REGION Network 1: Block description — Sections 1 to 2
   // ▄▄▄▄▄▄▄▄▄▄▄▄▄▄▄▄▄▄▄▄▄▄▄▄▄▄▄▄▄▄▄▄▄  ＳＴＡＮＤＡＲＤ  ▄▄ 
   // 
   // 
   // TITLE:    DEVICE DRIVER — THREE-WAY VALVE
   // 
   // 
   // ▀▀▀▀▀▀▀▀▀▀▀▀▀▀▀▀▀▀▀▀▀▀▀▀▀▀▀▀▀▀▀▀▀▀▀▀▀▀▀▀▀▀▀▀ 
   // 
   // ┌──────────────────────────────────────────┐
   // │                                          │
   // │          FC11011 — SOFTWARE MODULE DESIGN SPECIFICATION (SMDS)            │
   // │                                          │
   // │      The PDF version of the SMDS for this module is available online here:        │
   // │              https://psop.uk/pal-smds-fc11011-p               │
   // │                                          │
   // │      It is also available as part of the Project User Defined Documentation,      │
   // │      it can be accessed by selecting this module in the Project Tree          │
   // │      (on the left) and pressing SHIFT+F1                        │
   // │                                          │
   // └─────────────────────────────────────── ʷᴵᴰ⁻ᵇᶠᵍ  ┘
   // 
   // FC11011_StdDevValve3Way controls the operation of 3-way valve with a common energised port 
   // (the action of the valve switches the common port to one of the other two ports) configured with 
   // either position feedback or no position feedback.
   // 
   // The module supports automatic and manual control and can be configured with simulation mode 
   // to allow the valve limit switch signals to be overwritten and set to follow the demand output. 
   // 
   // The module generates fault logic for the valve that will trigger specific alarms depending on the 
   // fault in question. The alarms within this block are: 
   // 
   //    •   Failed to Energise 
   // 
   //    •   Failed to Deenergise 
   // 
   //    •   Failed while Energised
   // 
   //    •   Failed while Deenergised
   // 
   //    •   External Fault 
   // 
   // Separate operation times for energising and deenergising can be defined. 
   // 
   // The valve module supports all forms of interlock, permissive and trip signals, and emergency stop 
   // signals. The module has the conditional facility to allow the operator to bypass interlocks, 
   // permissive and trip conditions.
   // 
   // Various status signals are generated for supervisory systems:
   // 
   //    •   Deenergised
   // 
   //    •   Energising
   // 
   //    •   Energised
   // 
   //    •   Deenergising
   // 
   //    •   Fault
   // 
   // The module also generates status signals for the selected operating modes and conditions.
   // 
   // 
   // ▄▄▄▄▄▄▄▄▄▄▄▄▄▄▄▄▄▄▄▄▄▄▄▄▄▄▄▄▄▄▄▄▄▄▄▄▄▄▄▄▄▄▄▄
   // 1.     BLOCK TECHNICAL SUMMARY
   // 
   // 
   //  ――――――――――――――――――――――――――――――――――――――――――
   //  NOMENCLATURE & ADDRESSING
   //  ――――――――――――――――――――――――――――――――――――――――――
   //  BLOCK TITLE         Three-way Valve
   //  BLOCK FUNCTION GROUP    Device Driver 
   //  BLOCK ADDRESS       FC11011
   //  BLOCK SYMBOL        FC11011_StdDevValve3Way
   //  BLOCK USER ID         StdDevValve3Way
   // 
   //  ――――――――――――――――――――――――――――――――――――――――――
   //  BLOCK TYPE & USAGE
   //  ――――――――――――――――――――――――――――――――――――――――――
   //  BLOCK TYPE         Function (FC)
   //  BLOCK NUMBER        11011
   //  LANGUAGE           LAD
   //  OPTIMISED ACCESS     Yes
   //  PAL USAGE TYPE       Standard block
   // 
   //  ――――――――――――――――――――――――――――――――――――――――――
   //  METRICS
   //  ――――――――――――――――――――――――――――――――――――――――――
   //  EXECUTION TIME       66.5 μs¹
   //  LOAD MEMORY       98.6 kB
   //  WORK MEMORY           2.1 kB  
   //  ――――――――――――――――――――――――――――――――――――――――――
   //                ¹ Measured on: CPU-1515-2PN (order no. 6ES7512-2AM02-0AB0) 
   //                             https://psop.uk/pal-ds-cpu1515
   // 
   // 
   // 
   // ▂▂▂▂▂▂▂▂▂▂▂▂▂▂▂▂▂▂▂▂▂▂▂▂▂▂▂▂▂▂▂▂▂▂▂▂▂▂▂▂▂▂▂▂
   // 1.1      Additional document references
   // 
   // 
   // Only those documents specified in OB1 (section DOCUMENT REFERENCES) are listed within this 
   // block. There are no additional document references.
   // 
   //                ━━━   ⬙⬙⬙⬙⬙⬙   ━━━
   // 
   // 
   // 
   // ▄▄▄▄▄▄▄▄▄▄▄▄▄▄▄▄▄▄▄▄▄▄▄▄▄▄▄▄▄▄▄▄▄▄▄▄▄▄▄▄▄▄▄▄
   // 2.     FUNCTIONAL DESCRIPTION
   // 
   // 
   // FC11011 is the Three Way Valve block, it is a comprehensive block designed to operate and 
   // monitor a standard three-way valve.
   // 
   // 
   // 
   // ▂▂▂▂▂▂▂▂▂▂▂▂▂▂▂▂▂▂▂▂▂▂▂▂▂▂▂▂▂▂▂▂▂▂▂▂▂▂▂▂▂▂▂▂
   // 2.1     Defining a three-way valve
   // 
   // 
   // A three-way (or diverting) valve is any valve that can connect a common port to one of two other 
   // ports, depending on its energised state:
   // 
   // 
   //        DEENERGISED STATE              ENERGISED STATE
   //                             ⣀⣴⠶⠛⠛⠛⠷⢦⣄                                                         ⣠⡴⠶⠛⠛⠛⠶⣦⣄                            
   //                         ⢀⡾⠋              ⠙⢷⡄                                                 ⢠⡾⠋              ⠙⢷⡀                        
   //                         ⣾⠁                    ⢿⡀                                               ⣿⠁                  ⠈⣷                        
   // ⣼⣿⣿⣿⣿⣷⣤⡀        ⣿⠛⠛⠛⠛⠛⣿          ⣸⠇        ⣠⡾⠛⠛⠛⠛⣷ ⣾⣿⣿⣿⣿⣷⣄⡀      ⠸⣿⠛⠛⠛⠛⠛⣿          ⣿        ⢀⣠⣾⣿⣿⣿⣿⣷
   // ⣿⣿⣿⣿⣿⣿⣿⣿⣶⣄    ⢹⣆        ⣿        ⢠⡿    ⣀⣴⠟⠁          ⣿ ⣿⣿⣿⣿⣿⣿⣿⣿⣦⣄    ⢻⡄        ⣿        ⣰⡟    ⣠⣴⣿⣿⣿⣿⣿⣿⣿⣿
   // ⣿⣿⣿⣿⣿⣿⣿⣿⣿⣿⣿⣦⣀⠙⢷⣄⡀  ⣿    ⣀⣴⠟⢀⣤⠞⠋                ⣿ ⣿⣿⣿⣿⣿⣿⣿⣿⣿⣿⣷⣦⡀⠻⢦⣄    ⣿  ⢀⣠⡾⠋⢀⣴⣿⣿⣿⣿⣿⣿⣿⣿⣿⣿⣿
   // ⣿⣿⣿⡿⠛⣉⣠⣤⣉⠙⠻⣿⣿⣷⣤⡉⠙⠛⣿⠛⠛⠉⣠⡾⠋⠁                    ⣿ ⣿⣿⣿⡿⠋⣉⣤⣤⣉⠙⢿⣿⣿⣷⣄⡉⠛⠛⣿⠛⠛⢉⣤⣾⣿⣿⣿⣿⣿⣿⣿⣿⣿⣿⣿⣿⣿
   // ⣿⣿⡏⢠⣾⣿⣿⣿⣿⣿⣆⠘⣿⣿⣿⣿⣶⣄⣿⣠⡴⠟⠁                          ⣿ ⣿⣿⠏⢠⣿⣿⣿⣿⣿⣿⡄⠹⣿⣿⣿⣿⣦⣄⣿⣠⣴⣿⣿⣿⣿⣿⣿⣿⣿⣿⣿⣿⣿⣿⣿⣿⣿
   // ⣿⣿  ⣿⣿⣿⣿⣿⣿⣿⣿  ⣿⣿⣿⣿⣿⣿⣿⡋                                ⣿ ⣿⣿  ⣿⣿⣿⣿⣿⣿⣿⣿  ⣿⣿⣿⣿⣿⣿⣿⣿⣿⣿⣿⣿⣿⣿⣿⣿⣿⣿⣿⣿⣿⣿⣿⣿⣿
   // ⣿⣿⣇⠘⢿⣿⣿⣿⣿⣿⠏⢠⣿⣿⣿⣿⣿⣿⣿⣿⣷⣄⡀                          ⣿ ⣿⣿⣆⠹⣿⣿⣿⣿⣿⣿⠏⣰⣿⣿⣿⣿⣿⡟⠉⢿⣿⣿⣿⣿⣿⣿⣿⣿⣿⣿⣿⣿⣿⣿⣿⣿⣿
   // ⣿⣿⣿⣷⣄⣉⠛⠛⢋⣡⣴⣿⣿⣿⢟⣽⣿⣿⣿⣿⣿⣿⡛⢶⣄                      ⣿ ⣿⣿⣿⣷⣄⣉⠛⠛⣉⣠⣾⣿⣿⡿⢟⡿⠋      ⠙⣯⡻⣿⣿⣿⣿⣿⣿⣿⣿⣿⣿⣿⣿⣿⣿
   // ⣿⣿⣿⣿⣿⣿⣿⣿⣿⣿⣿⠿⠋⣠⣿⣿⣿⣿⣿⣿⣿⣿⣿⣦⠉⠻⣦⣀                ⣿ ⣿⣿⣿⣿⣿⣿⣿⣿⣿⣿⣿⠟⠉⣰⠟⠁          ⠈⢻⣄⠙⠻⣿⣿⣿⣿⣿⣿⣿⣿⣿⣿⣿
   // ⣿⣿⣿⣿⣿⣿⣿⣿⡿⠛⠁⢀⣼⣿⣿⣿⣿⣿⣿⣿⣿⣿⣿⣿⣷⡄  ⠙⠷⣤⡀          ⣿ ⣿⣿⣿⣿⣿⣿⣿⣿⠿⠋  ⢠⡾⠃                  ⠙⢷⡀⠈⠙⢿⣿⣿⣿⣿⣿⣿⣿⣿
   // ⢻⣿⣿⣿⣿⡿⠟⠁    ⣰⣿⣿⣿⣿⣿⣿⣿⣿⣿⣿⣿⣿⣿⣿⣿⣦⡀  ⠈⠙⢶⣤⣤⣤⣤⡿ ⢿⣿⣿⣿⣿⡿⠋⠁    ⣴⠟                        ⠈⠻⣦    ⠈⠛⢿⣿⣿⣿⣿⡿
   //                 ⢀⣾⣿⣿⣿⣿⣿⣿⣿⣿⣿⣿⣿⣿⣿⣿⣿⣿⣿⣿⣄                                 ⣠⡾⠁                              ⠘⢷⡄                
   //               ⣰⣿⣿⣿⣿⣿⣿⣿⣿⣿⣿⣿⣿⣿⣿⣿⣿⣿⣿⣿⣿⣿⣧                             ⣴⠏                                      ⠹⣦              
   //               ⣿⣿⣿⣿⣿⣿⣿⣿⣿⣿⣿⣿⣿⣿⣿⣿⣿⣿⣿⣿⣿⣿⣿                             ⣿                                          ⣿              
   //               ⠻⣿⣿⣿⣿⣿⣿⣿⣿⣿⣿⣿⣿⣿⣿⣿⣿⣿⣿⣿⣿⣿⡿                             ⢿⣤⣤⣤⣤⣤⣤⣤⣤⣤⣤⣤⣤⣤⣤⣤⣤⣤⣤⣤⣤⣤⡟              
   // 
   //   Common port (left) connected to bottom port     Common port (left) connected to right port
   // 
   // 
   // The left-hand image above shows a three-way valve in a deenergised state, the common port 
   // (on the left, signified by the circle on a dark background) is connected to port 1 (the bottom port, 
   // or the deenergised port). If the valve is energised (voltage is applied to its solenoid), the 
   // common port now becomes connected to port 2 (on the right, or the energised port), right-hand 
   // image.
   // 
   // Like the isolating valve (controlled by FC11001), the three-way valve has only two states, it is 
   // either deenergised to port 1 or energised to port 2 and cannot sustain any intermediate position. 
   // Three-way valves are generally spring-return type valves that adopt a particular state when 
   // energised, and return to the other state when deenergised. Such valves are generally operated 
   // directly via an electronic solenoid. Some are pneumatically operated, again by activating a 
   // solenoid that when energised applies air to one side to the valve, driving it to the energised 
   // state, the solenoid then vents the air when deenergised allowing the valve to return to its 
   // deenergised state via the spring-return mechanism within the valve. 
   // 
   // Three-way valves have a single flow-path through the valve, and this path either connects the 
   // common port to the deenergised port or to the energised port. Unlike the isolating valve (that is 
   // either energised or deenergised), the three-way valve is never deenergised, the common port 
   // will always be connected to one of the other ports and there will always be a flow path through 
   // the valve.
   // 
   // Three-way valves have many different orientations and left/right, top/bottom configurations, these 
   // can be seen in Appendix A of the SMDS, available here:
   // 
   //      https://psop.uk/pal-smds-fc11011-p
   // 
   // In the above symbols, the lines in the actuator circle at the top of the symbol show, 
   // schematically, the flow path when the valve is deenergised, i.e. it shows which two ports are 
   // open when the valve is deenergised.
   // 
   // 
   // 
   // ▂▂▂▂▂▂▂▂▂▂▂▂▂▂▂▂▂▂▂▂▂▂▂▂▂▂▂▂▂▂▂▂▂▂▂▂▂▂▂▂▂▂▂▂
   // 2.1.1     Comparison with an isolating valve
   // 
   // 
   // From a software perspective, the thee-way valve and the isolating valve are very similar, both 
   // change state when an output signal is energised and both may be equipped with limit switches 
   // to positively identify the state of the valve.
   // 
   // Both the isolating valve and the three-way valve have operation timers that activate whenever 
   // the valve changes state and both generate faults in much the same way.
   // 
   // The main difference between a three-way valve and an isolating valve, is that the three-way 
   // valve does not have normally open and normally closed¹ types. Three-way valves are always 
   // open — the common port will always be connected to one of the other ports, hence the normally 
   // open/closed operation is simply determined by how the valve is physically connected to the 
   // pipework and how the deenergised state of the valve is orientated. Symbolically, each 
   // configuration of the valve is supported and an appropriate symbol is available for all 
   // orientations, see Appendix A of the SMDS, available here:
   // 
   //      https://psop.uk/pal-smds-fc11011-p
   // 
   // Where an isolating valve uses the terms OPEN and CLOSED &c. the three-way valve uses the 
   // terms ENERGISED and DEENERGISED; the direct comparisons are as follows:
   // 
   // 
   //  ――――――――――――――――――――――――――――――――――――――――――
   //  ISOLATING VALVE TERMINOLOGY       THREE-WAY VALVE TERMINOLOGY
   //  ――――――――――――――――――――――――――――――――――――――――――
   //  Closed                    Deenergised
   //  Opening                   Energising
   //  Open                   Energised
   //  Closing                   Deenergising
   //  ――――――――――――――――――――――――――――――――――――――――――
   // 
   // 
   // ――――――――――
   // ¹         For an isolating valve, normally closed refers to a valve that is deenergised in the 
   //      closed state and will open when an energising signal is applied. A normally open 
   //      valve operates in the reverse arrangement, the valve is open in the deenergised 
   //      state and will only close when the energising signal is present. Normally open valves 
   //      are used in fail-safe applications where a power failure causes the valve to open by 
   //      default, usually to vent pressure or release some other motive force from the vessel 
   //      to which it is connected.
   // ――――――――――
   // 
   // 
   //                      
   // ▂▂▂▂▂▂▂▂▂▂▂▂▂▂▂▂▂▂▂▂▂▂▂▂▂▂▂▂▂▂▂▂▂▂▂▂▂▂▂▂▂▂▂▂
   // 2.1.2     Valve operating times
   // 
   // 
   // A three-way valve, will move from its deenergised state to its energised state when the operating 
   // signal is applied; this transition will occur in a specified time (the time taken will depend on the 
   // size and operating mechanism within the valve itself), this is referred to as the energising 
   // operation time.
   // 
   // Similarly, the transition from energised to deenergised will again occur in a specified time. This 
   // is referred to as the deenergising operation time. 
   // 
   // The energising and deenergising times can be different for a given valve. 
   // 
   // Collectively, the energising and deenergising times are referred to as the operating times 
   // (sometimes operation times) of the valve.
   // 
   // The maximum energising and deenergising times for a valve are generally given as part of the 
   // specification for the valve itself.
   // 
   // If a valve does not reach the required state within the specified maximum operating times, the 
   // valve is generally considered to be in a fault condition (either failed to energise or failed to 
   // deenergise depending on the action being undertaken).
   // 
   // 
   // 
   // ▂▂▂▂▂▂▂▂▂▂▂▂▂▂▂▂▂▂▂▂▂▂▂▂▂▂▂▂▂▂▂▂▂▂▂▂▂▂▂▂▂▂▂▂
   // 2.1.3     Valve position feedback arrangements
   // 
   // 
   // Three-way valves can be equipped with limit switch signals that positively identify the current 
   // position of the valve. There are four combinations of limit switches:
   // 
   //    1.  No limit switches         There is no positive indication of the current state 
   //                      of the valve, it is assumed to be in the expected 
   //                      state.
   // 
   //    2.  Deenergised limit switch only     Positive indication is given for the deenergised 
   //                      state only. The valve is assumed to be in the 
   //                      energised state if the deenergised signal is 
   //                      inactive.
   // 
   // 
   //    3.  Energised limit switch only       Positive indication is given for the energised 
   //                      state only. The valve is assumed to be 
   //                      deenergised if the energised signal is inactive.
   // 
   // 
   //    4.  Energised and deenergised        Positive indication is given for both states. 
   //      limit switches            This allows the true state of the valve to be 
   //                      determined under all circumstances.
   // 
   // 
   // Note:    Positive indication of a valve state need not be determined by a limit switch (though this 
   //      is by far the most common arrangement), it could for example, be determined by some 
   //      process value: if a flow is detected after the energising of a valve, for example.
   // 
   //      In practice, limit switches are the preferred mechanism for the positive indication 
   //      of a given valve state.
   // 
   // Where a limit switch is absent, the valve is assumed to have reached the correct position when 
   // the relevant operation time has counted for an adjustable percentage of its maximum operating 
   // time.
   // 
   // 
   // 
   // ▂▂▂▂▂▂▂▂▂▂▂▂▂▂▂▂▂▂▂▂▂▂▂▂▂▂▂▂▂▂▂▂▂▂▂▂▂▂▂▂▂▂▂▂
   // 2.2     Module operation
   // 
   // 
   // FC11011 is used to control (operate) a three-way valve, the module also monitors the various 
   // configurations of valve position feedback signals to determine if the valve is in a fault condition.
   // 
   // The module will drive the valve to the requested state by energising or deenergising a digital 
   // signal (usually a digital output signal).
   // 
   // If the requested state of the valve requires the output to be energised, the output will remain 
   // energised until the requested state changes.
   // 
   // If the requested state signal changes (either from deenergised to energised, or from energised 
   // to deenergised), the module will start either an energising operation timer (request has changed 
   // from deenergised to energised) or a deenergising operation timer (request has changed from 
   // energised to deenergised); these timers can have different values.
   // 
   // The valve will be expected to reach the requested state before the relevant operation timer 
   // expires; if it does not, the valve will enter a fault state and an appropriate alarm will be generated 
   // when the operation timer expires.
   // 
   // Once the valve has reached its requested state, the operation time will reset and the module 
   // will continue to monitor the state of the valve. 
   // 
   // If the request signal changes whilst the valve is in the process of changing state (e.g. the valve is 
   // requested to change from deenergised to energised and whilst the energising operation timer is 
   // running, the request is changed back to deenergised), the running operation timer will be reset 
   // and the operation timer for the second request will start from its specified value. I.e. no 
   // allowance is made for how far the valve may have moved following the first request change.
   // 
   // If the valve is stable, in a given state (i.e. is not in the process of changing state) and the valve 
   // position signals no longer match the required state (e.g. the valve had correctly energised, but 
   // at some time after this, the energised position feedback is lost), the valve will instantly generate 
   // an alarm condition.
   // 
   // 
   // 
   // ▂▂▂▂▂▂▂▂▂▂▂▂▂▂▂▂▂▂▂▂▂▂▂▂▂▂▂▂▂▂▂▂▂▂▂▂▂▂▂▂▂▂▂▂
   // 2.3     Safety and interlocks
   // 
   // 
   // The module, optionally, accommodates a single safety signal (emergency stop), and the 
   // standard arrangement of up to three interlock signals (interlock, permissive and trip) as follows:
   // 
   // 
   // 
   // ▂▂▂▂▂▂▂▂▂▂▂▂▂▂▂▂▂▂▂▂▂▂▂▂▂▂▂▂▂▂▂▂▂▂▂▂▂▂▂▂▂▂▂▂
   // 2.3.1     Safety (emergency stop) signal
   // 
   // 
   // Safety or emergency stop signals are hardwired signals that remove power from a device forcing 
   // it to a safe state. Such signals act independently of the software (the pressing of an emergency 
   // stop button will physically remove power from the affected devices).
   // 
   // The emergency stop signal passed to the module is used to allow the state of the valve to be 
   // correctly interpreted within the software under emergency stop conditions.
   // 
   // When the emergency stop signal is removed, the valve will resume the requested state (with 
   // the appropriate operation timer).
   // 
   // The presence of an emergency stop signal is indicated via the block icon status signals 
   // generated by the module (see §§ 2.7 and 4).
   // 
   // Emergency stop signals cannot be bypassed under any circumstances (cf. interlock signals, 
   // below).
   // 
   // 
   // 
   // ▂▂▂▂▂▂▂▂▂▂▂▂▂▂▂▂▂▂▂▂▂▂▂▂▂▂▂▂▂▂▂▂▂▂▂▂▂▂▂▂▂▂▂▂
   // 2.3.2     Interlock signals
   // 
   // 
   // There are three types of interlock signal:
   // 
   //    1.  Interlock
   //      A simple interlock that is active whenever a set of conditions is true; if active, it will 
   //      force the devices to a specified state.
   // 
   // 
   //    2.  Permissive
   //      Designates a specified “permitted” state for the device. A permissive interlock takes 
   //      no action if the device is in the non-permitted state, but once the device changes to 
   //      the permitted state, it will be prevented from changing back to the non-permitted state 
   //      (e.g. if the permitted state was deenergised and the valve was currently energised 
   //      when the permissive signal activated, it would not force the valve to deenergised, 
   //      but once it was deenergised, it would prevent it from re-energising).
   // 
   //    3.  Trip
   //      A latching interlock, it activates whenever a set of events are true (like an interlock), 
   //      but will not deactivate until the triggering conditions are removed and a reset signal 
   //      has been given (effectively a latching interlock); if active, it will force the device to a 
   //      specified state.
   // 
   // Note:    The trip reset signal is handled by the trip logic, the valve module will simply respond 
   //      to the presence or absence of a trip signal.
   // 
   // Each type of interlock has its own individual signal passed to the module (three signals in total).
   // 
   // Interlock signals can be optionally bypassed (effectively disabled) under specific, manually 
   // selected operations.
   // 
   // 
   // 
   // ▂▂▂▂▂▂▂▂▂▂▂▂▂▂▂▂▂▂▂▂▂▂▂▂▂▂▂▂▂▂▂▂▂▂▂▂▂▂▂▂▂▂▂▂
   // 2.3.3     Priority of safety and interlock signals
   // 
   // 
   // The presence of any interlock stop signal is indicated via the block icon status signals generated 
   // by the module (see § 4). The priority order of the various types of interlock (if more than one is 
   // active at the same time) is as follows:
   // 
   // 
   //  ――――――――――――――――――――――――――――――――――――――――――
   //  SIGNAL TYPE        PRIORITY        CAN BE BYPASSED
   //  ――――――――――――――――――――――――――――――――――――――――――
   //  Emergency Stop         High               NO
   //  Trip             ↑              YES
   //  Interlock             ↑              YES
   //  Permissive          Low               YES
   //  ――――――――――――――――――――――――――――――――――――――――――
   //  High priority signal take precedence over lower priority signals.
   // 
   // 
   // 
   // ▂▂▂▂▂▂▂▂▂▂▂▂▂▂▂▂▂▂▂▂▂▂▂▂▂▂▂▂▂▂▂▂▂▂▂▂▂▂▂▂▂▂▂▂
   // 2.4     Alarms and warnings
   // 
   // 
   // The module can generate up to five distinct alarms:
   // 
   // 
   //    1.  FAILED TO ENERGISE
   //      Indicates that the valve did not energise when requested to do so. The alarm is 
   //      generated when the energising operation timer expires without the corresponding 
   //      position feedback activating.
   // 
   // 
   //    2.  FAILED TO DEENERGISE
   //      Indicates that the valve did not deenergise when requested to do so. The alarm is 
   //      generated when the deenergising operation timer expires without the corresponding 
   //      position feedback activating.
   // 
   // 
   //    3.  FAILED WHILE ENERGISED
   //      Indicates that the valve energised correctly, but then at some later point, the position 
   //      feedback signals, indicating the energised state of the valve, were lost.
   // 
   //      
   //    4.  FAILED WHILE DEENERGISED
   //      Indicates that the valve deenergised correctly, but then at some later point, the position 
   //      feedback signals, indicating the deenergised state of the valve, were lost
   // 
   // 
   //    5.  EXTERNAL FAULT
   //      External fault is a separate (and optional) hardwired signal from the valve that 
   //      indicates the valve itself has detected a problem (e.g. a trip signal from a 
   //      motorised valve)
   // 
   // The module does not generate any warnings.
   // 
   // 
   // 
   // ▂▂▂▂▂▂▂▂▂▂▂▂▂▂▂▂▂▂▂▂▂▂▂▂▂▂▂▂▂▂▂▂▂▂▂▂▂▂▂▂▂▂▂▂
   // 2.4.1     Alarm — Failed to energise/deenergise
   // 
   // 
   // Failed to energised and failed to deenergised alarms are generated if the valve is required to 
   // change state and fails to do so within the time set by the relevant operation timer.
   // 
   // For example, if the valve were in a deenergised state and was requested to energised, the failed 
   // to energised alarm would be generated if the valve had not received positive indication that the 
   // valve was correctly energised (from the valve limit switches) by the time the energising 
   // operation timer expired.
   // 
   // If the valve is not equipped with any limit switches, then there are no circumstances under 
   // which the failed to energised and failed to deenergised alarms can be generated (the valve is 
   // always assumed to operate correctly and be in the required position).
   // 
   // 
   // 
   // ▂▂▂▂▂▂▂▂▂▂▂▂▂▂▂▂▂▂▂▂▂▂▂▂▂▂▂▂▂▂▂▂▂▂▂▂▂▂▂▂▂▂▂▂
   // 2.4.2     Alarm — Failed while energised/deenergised
   // 
   // Failed while  energised and failed while deenergised are generated if the valve is in a steady 
   // state (not in the process of changing from energised to deenergised or vice versa) and the 
   // positive indication of the valve position changes to indicate the steady state position has 
   // changed.
   // 
   // An example would be for valve with both energised and deenergised limit switches, to be in the 
   // energised state, where the energised limit is active and deenergised limit is inactive (positively 
   // indicating the valve is energised). If the power to the valve failed (a blown fuse or broken wire, 
   // for example), the valve would deenergise and return to the deenergised state and this would be 
   // reflected in the state of the limit switches. The module, knowing nothing of the power failure, 
   // would expect the valve to still be energised and would instantly generate a failed while energised 
   // alarm.
   // 
   // If the valve is not equipped with any limit switches, then there are no circumstances under which 
   // the failed while energised and failed while deenergised alarms can be generated (the valve is 
   // always assumed to operate correctly and be in the required position).
   // 
   // 
   // 
   // 
   // ▂▂▂▂▂▂▂▂▂▂▂▂▂▂▂▂▂▂▂▂▂▂▂▂▂▂▂▂▂▂▂▂▂▂▂▂▂▂▂▂▂▂▂▂
   // 2.4.3     Alarm — External fault
   // 
   // 
   // The external fault alarm is activated whenever the external fault signal provided to the module 
   // is active. The external fault signal is an optional signal that indicates that the valve itself is 
   // experiencing a problem. The signal is more commonly associated with motorised valves where 
   // thermal overload signals are used to indicate that the valve motor has experienced a fault, 
   // it could also be used to indicate the loss of pneumatic pressure for pneumatic solenoid valves.
   // 
   // 
   // 
   // ▂▂▂▂▂▂▂▂▂▂▂▂▂▂▂▂▂▂▂▂▂▂▂▂▂▂▂▂▂▂▂▂▂▂▂▂▂▂▂▂▂▂▂▂
   // 2.4.4     Resetting alarm conditions
   // 
   // 
   // The four alarms derived from valve position feedback signals:
   // 
   //    1.  FAILED TO ENERGISE
   // 
   //    2.  FAILED TO DEENERGISE
   // 
   //    3.  FAILED WHILE ENERGISED
   // 
   //    4.  FAILED WHILE DEENERGISED
   // 
   // Are latching alarms, if the alarm conditions occur, the valve will be placed in a fault condition 
   // (see § 2.5) and will no longer be operable, the valve will remain in a deenergised condition until 
   // the fault is corrected.
   // 
   // The alarm conditions are only reset when the module receives a RESET command (usually 
   // from the operator).
   // 
   // The fifth alarm:
   // 
   //    5.  EXTERNAL FAULT
   // 
   // Is a non-latching alarm that is reset automatically whenever the external fault signal is 
   // deactivated. It should be noted however, that the cause of the external fault (say a thermal 
   // overload) may itself, require some form of manual or physical reset, before the fault condition 
   // is removed.
   // 
   // 
   // 
   // ▂▂▂▂▂▂▂▂▂▂▂▂▂▂▂▂▂▂▂▂▂▂▂▂▂▂▂▂▂▂▂▂▂▂▂▂▂▂▂▂▂▂▂▂
   // 2.5     Fault conditions
   // 
   // 
   // The valve is in a fault condition if any alarm conditions is active:
   // 
   //    1.  FAILED TO ENERGISE
   // 
   //    2.  FAILED TO DEENERGISE
   // 
   //    3.  FAILED WHILE ENERGISED
   // 
   //    4.  FAILED WHILE DEENERGISED
   // 
   //    5.  EXTERNAL FAULT
   // 
   // A valve cannot operate if any fault condition is active and it will return to its deenergised state.
   // 
   // A valve that is in a fault state will ignore any request that would move it to an energised state, 
   // irrespective of the source of the command: automatic operation, manual operation or even an 
   // interlock condition.
   // 
   // 
   // 
   // ▂▂▂▂▂▂▂▂▂▂▂▂▂▂▂▂▂▂▂▂▂▂▂▂▂▂▂▂▂▂▂▂▂▂▂▂▂▂▂▂▂▂▂▂
   // 2.6     Operating modes
   // 
   // 
   // The module supports the following optional modes of operation:
   // 
   //    •   Automatic/manual mode (allows the operator to take manual control of the valve 
   //      and energise or deenergise it irrespective of the control system requirements)
   // 
   //    •   Interlock bypass mode (allows the operator to override permissive, interlock and 
   //      trip signals
   // 
   //    •   Simulation mode (allows the operator to override the current instrument position 
   //      feedback signals with simulated values)
   // 
   //    •   Remote/local/all selection (allows control of the instrument to be restricted to a 
   //      specific SCADA/HMI device) 
   // 
   //    •   Faceplate disabled (informs the supervisory system not to display any faceplates 
   //      for the device, preventing graphical operator selections)
   // 
   // 
   // 
   // ▂▂▂▂▂▂▂▂▂▂▂▂▂▂▂▂▂▂▂▂▂▂▂▂▂▂▂▂▂▂▂▂▂▂▂▂▂▂▂▂▂▂▂▂
   // 2.6.1     Automatic and manual control modes
   // 
   // 
   // By default, the module will be in automatic mode; this means that any energise or deenergise 
   // instruction received by the module from the control software (continuous or sequential control) 
   // will cause the valve to adopt the requested state (if the valve is not in fault and is free of 
   // interlock and safety conditions).
   // 
   // If the module is switched to manual mode, the automatic control signals will be ignored and the 
   // module will adopt the state required by the manual request signals set by the operator 
   // (again, the valve must not be in fault and must be free of interlock and safety conditions).
   // 
   // Selecting automatic or manual mode is an operator action and can be implemented at any time. 
   // Changing from automatic mode to manual mode is a bumpless operation, in which the initial 
   // manual state of the valve is set to match the current automatic state. For example, if a valve 
   // were energised under automatic control, switching the valve to manual would cause the initial 
   // manual state to be set to energised (matching the automatic state), ensuring that the valve does 
   // not initially change state when changing to manual mode.
   // 
   // Once manual mode is established, the operator is free to energise and deenergise the valve 
   // as required.
   // 
   // There is no bumpless transfer back to automatic mode, the valve will simply adopt the state 
   // required by the control software.
   // 
   // Interlocks and safety signals operate in exactly the same way for a valve in manual mode 
   // as they do for a valve in automatic mode and will take priority over any command issued in either 
   // automatic or manual mode.
   // 
   // 
   // 
   // ▂▂▂▂▂▂▂▂▂▂▂▂▂▂▂▂▂▂▂▂▂▂▂▂▂▂▂▂▂▂▂▂▂▂▂▂▂▂▂▂▂▂▂▂
   // 2.6.2     Interlock bypass mode
   // 
   // 
   // Interlock bypass mode allows the three interlock types (trip, interlock and permissive) to be 
   // overridden (bypassed) by the operator.
   // 
   // If bypass mode is activated, any interlock signal will be ignored by the module.
   // 
   // Bypass mode is an entirely manual operation that can only be initiated by an operator, usually 
   // via a supervisory system (SCADA or HMI).
   // 
   // 
   // 
   // ▂▂▂▂▂▂▂▂▂▂▂▂▂▂▂▂▂▂▂▂▂▂▂▂▂▂▂▂▂▂▂▂▂▂▂▂▂▂▂▂▂▂▂▂
   // 2.6.3     Simulation mode
   // 
   // 
   // The module can be switched to a simulation mode, under which any positive position feedback 
   // signals from valve limit switches are replaced by simulated signals selected by the operator. 
   // Simulation mode can be used during testing and can also be applied in a process environment 
   // if a fault condition is detected within the valve.
   // 
   // The operator can select any one of the following possible simulation arrangements (only one 
   // can be active at any given time):
   // 
   // 
   //    •   Follow demand    The simulation will generate energised and deenergised 
   //                 feedback signals that match the requested state of the valve
   // 
   //    •   Energised        The simulation will generate signals to give a permanently 
   //                 energised state for the valve, irrespective of any valve state 
   //                 request (allows failed to energised conditions to be 
   //                 simulated)
   // 
   //    •   Deenergised         The simulation will generate signals to give a permanently 
   //                 deenergised state for the valve, irrespective of any valve 
   //                 state request (allows failed to deenergised conditions to be 
   //                 simulated)
   // 
   //    •   No limits       No position feedback signals will be simulated
   // 
   // Simulation mode is a manual operation that can only be initiated by an operator.
   // 
   // 
   // 
   // ▁▁▁▁▁▁▁▁▁▁▁▁▁▁▁▁▁▁▁▁▁▁▁▁▁▁▁▁▁▁▁▁▁▁▁▁▁▁▁▁▁▁▁▁
   // 2.6.4     Remote/local/all mode
   // 
   // Remote and local operating modes refer to the device that has control of the module; where 
   // a plant has more than one SCADA/HMI, say a SCADA in a remote control room and a field 
   // mounted HMI local to the device, it is possible to restrict the operator control of the module to 
   // one, or the other, or both supervisor systems as follows
   // 
   //    •   Remote Only the remote system in the control room can control the device
   // 
   //    •   Local     A local system has taken control of the device and the remote system can 
   //            no longer issue commands to it
   // 
   //    •    All    Any system can control the device
   // 
   // The default arrangement if for all systems to have access to the device.
   // 
   // 
   // 
   // ▁▁▁▁▁▁▁▁▁▁▁▁▁▁▁▁▁▁▁▁▁▁▁▁▁▁▁▁▁▁▁▁▁▁▁▁▁▁▁▁▁▁▁▁
   // 2.6.5     Faceplate disabled mode
   // 
   // Prevents the supervisory system from displaying the faceplate from which the above options are 
   // selected. If the faceplate is disabled, the operator will not be able to select or change any of the 
   // various operating modes.
   // 
   // 
   // 
   // ▁▁▁▁▁▁▁▁▁▁▁▁▁▁▁▁▁▁▁▁▁▁▁▁▁▁▁▁▁▁▁▁▁▁▁▁▁▁▁▁▁▁▁▁
   // 2.7      Supervisory system interface
   // 
   // See the online documentation for this block — select the block in the project tree and press:
   //      SHIFT + F1 or follow the link: https://psop.uk/pal-smds-fc11011-p 
   // 
   // The supervisory system interface is available in sections 2.5 and 4 of the online SMDS 
   // document.
   // 
   //                ━━━   ⬙⬙⬙⬙⬙⬙   ━━━
END_REGION

REGION Network 2: Block description — Section 3 to 3.2
   // ▄▄▄▄▄▄▄▄▄▄▄▄▄▄▄▄▄▄▄▄▄▄▄▄▄▄▄▄▄▄▄▄▄▄▄▄▄▄▄▄▄▄▄▄
   // 3.     DETAILED BLOCK DESCRIPTION
   // 
   // 
   // This module, FC11011_StdDevValve3Way uses user data types to provide the primary interface 
   // to the module, it also uses direct digital signals to provide an interface for the position feedback 
   // signals and for the fault, safety and interlock signals. It also has a single output signal used to 
   // operate the valve. 
   // 
   // These are the formal module parameters: 
   // 
   //  ――――――――――――――――――――――――――――――――――――――――――
   //  PARAM         FUNCTION                    TYPE      IN-OUT 
   //  ――――――――――――――――――――――――――――――――――――――――――
   //  SYS_SIGNALS      Common system signals              UT21000    In
   //           logic and timing signals for parametric access
   // 
   //  FBK_ENG        Optional energised state positive feedback     Bool      In
   //           (1 = energised, 0 = not energised) If not 
   //           required, set permanently to _False
   // 
   //  FBK_DENG     Optional deenergised state positive feedback   Bool      In
   //           (1 = deenergised, 0 = not deenergised) If not  
   //           required, set permanently to _False
   // 
   //  EXT_FAULT     Optional external fault signal for the device     Bool      In
   //           (1 = fault, 0 = healthy). If not required, set 
   //           permanently to _False
   // 
   //  E_STOP        Optional emergency stop (safety) signal        Bool      In
   //           (1 = emergency stop active, 0 = healthy) If not 
   //           required, set permanently to _False
   // 
   //  TRIP        Optional trip signal                  Bool      In
   //           (1 = trip condition active, 0 = healthy) If not 
   //           required, set permanently to _False
   // 
   //  INTERLOCK     Optional interlock signal               Bool      In
   //           (1 = interlock condition active, 0 = healthy) If 
   //           not required, set permanently to _False
   // 
   //  PERMISSIVE      Optional permissive signal             Bool      In
   //           (1 = permissive condition active, 0 = healthy) 
   //           If not required, set permanently to _False
   // 
   //  STATIC_DATA     Data structure that holds the configuration data     UT11011    In
   //           for the device (limit switch and interlock 
   //           configuration &c.)
   // 
   //  DYNAMIC_DATA      Data structure that holds the live data for the       UT31011    InOut
   //           device (its mode, status and messages and 
   //           any other dynamic information required by the 
   //           module)
   // 
   //  OPERATE        Output to drive the valve to a particular state    Bool      Out
   //           (1 = energised state, 0 = deenergised state)
   //  ――――――――――――――――――――――――――――――――――――――――――
   // 
   // FBK_ENG, FBK_DENG and EXT_FAULT parameters are input signals provided directly from the 
   // device itself (via digital input cards). The OPERATE signal is an output signal (via a digital output 
   // card) that causes the valve to energised and deenergised.
   // 
   // The E-STOP parameter is the interface to any safety signal that might apply to the valve; 
   // similarly, the PERMISSIVE, INTERLOCK and TRIP parameters are the links to any such interlock 
   // signals that may be applied to the device.
   // 
   // The STATIC_DATA and DYNAMIC_DATA parameters are UDTs that hold (respectively) the 
   // configuration information and the live data for the device.
   // 
   //  ――――――――――――――――――――――――――――――――――――――――――
   //  PARAM         ASSOCIATED UDT          ASSOCIATED DATA BLOCK
   //  ――――――――――――――――――――――――――――――――――――――――――
   //  STATIC_DATA     UT11011_St_DevValve3Way        DB11011_St_DevValve3Way
   //  DYNAMIC_DATA   UT31011_Dy_DevValve3Way        DB31011_Dy_DevValve3Way
   //  ――――――――――――――――――――――――――――――――――――――――――
   // 
   // 
   // Section 6 contains a full list of all variables within these UDTs.
   // 
   // This arrangement conforms with the PAL philosophy where IO card connections, safety 
   // signals and interlocks have unique formal parameters; all remaining signals are passed as 
   // variables within UDTs, see the Software Design Specification [Ref. 008].
   // 
   // 
   // 
   // ▂▂▂▂▂▂▂▂▂▂▂▂▂▂▂▂▂▂▂▂▂▂▂▂▂▂▂▂▂▂▂▂▂▂▂▂▂▂▂▂▂▂▂▂
   // 3.1      Typical wiring arrangement
   // 
   // 
   // The typical wiring arrangements for a valve with all signals is as follows:
   // 
   //     24VDC  
   //      ─┬─                                ┌───────┐
   //       │                                 │       │  
   //       ├────┬────┐                 │      ─┴─
   //       │       │       │                 │        GND
   //       │       │       │             ┌┻┐ ▁▁
   //    ▁│ ○   ▁│○   ▁│○             │ │▁＼／ 
   //    ▔│ ○   ▔│○   ▔│○             │ │ ／＼   
   //     FAULT│     DENG│   ENG  │             └┬┘ ▔▔ 
   //       │   LIMIT │   LIMIT │                 │     
   //       │       │       │              │  
   //     ┌─┻─┐┌─┻─┐┌─┻─┐          ┌─┻─┐
   //     │  I1.0  ││  I1.1  ││  I1.2  │DI CARD        │  Q1.0 │DO CARD
   //     └─┬─┘└─┬─┘└─┬─┘          └─┬─┘
   //       │       │       │ ┌────────    │
   //       │       │       │ │ FC11011          │
   //       │       │       │ ├──────────┤ │
   //       │       │       │ │          │ │
   //       │       │       │ │           OPERATE ├─┘
   //       │       │       │ │          │
   //       │       │       └─┤ FBK_ENG          │
   //       │       │         │          │
   //       │       └──────┤ FBK_DENG           │
   //       │                 │          │
   //       └───────────┤ EXT_FAULT        │
   //                         │           
   //                         │
   // 
   // 
   // 
   // ▂▂▂▂▂▂▂▂▂▂▂▂▂▂▂▂▂▂▂▂▂▂▂▂▂▂▂▂▂▂▂▂▂▂▂▂▂▂▂▂▂▂▂▂
   // 3.2      Normal operation
   // 
   // 
   // Normal operation can generally be considered the operation of the valve under automatic or 
   // manual control (see § 3.6.1 for a full explanation of how automatic and manual modes are 
   // selected). And the mechanisms used to determine the state of the valve.
   // 
   // 
   // ▁▁▁▁▁▁▁▁▁▁▁▁▁▁▁▁▁▁▁▁▁▁▁▁▁▁▁▁▁▁▁▁▁▁▁▁▁▁▁▁▁▁▁▁
   // 3.2.1     Energising and deenergising the valve
   // 
   // 
   // Under automatic mode, the valve is controlled by separate software within the Controller (this 
   // is usually derived from either continuous control logic or sequential control logic and 
   // implemented by the command handling application module).
   // 
   // The result of this software will be to either energised the valve or deenergised the valve.
   // 
   // Under manual mode, the valve is controlled directly by the operator via some form of 
   // supervisory system (SCADA or HMI). Again, the result of the manual operator action will be to 
   // either energised or deenergised the valve.
   // 
   // There are two signals that, under normal operation, can cause the valve to move to a particular 
   // state, one for automatic mode and one for manual mode, both are passed to the module as 
   // part of the DYNAMIC_DATA parameter (UT31011_Dy_DevValve3Way):
   // 
   // 
   //  DATA STRUCTURE    UT31011_Dy_DevValve3Way
   //  ――――――――――――――――――――――――――――――――――――――――――
   //  SIGNAL         FUNCTION               TYPE     DETAILS
   //  ――――――――――――――――――――――――――――――――――――――――――
   //  ctrl_Aut_EngDeng    Causes the valve to energise and         Bool  1 = energise valve
   //            deenergise if automatic mode is        0 = deenergise valve
   //            active (mode_AutMan = 1). If auto
   //            mode is not active, signal is 
   //            ignored
   // 
   //  ctrl_Man_EngDeng   Causes the valve to energise and         Bool  1 = energise valve
   //            deenergise if manual mode is             0 = deenergise valve
   //            active (mode_AutMan = 0). If man
   //            mode is not active, signal is 
   //            ignored
   //  ――――――――――――――――――――――――――――――――――――――――――
   // 
   // The operating mode (either automatic or manual) is specified within the DYNAMIC_DATA 
   // parameter UDT (UT31011_Dy_DevValve3Way) mode_AutMan as follows:
   // 
   // 
   //  DATA STRUCTURE    UT31011_Dy_DevValve3Way
   //  ――――――――――――――――――――――――――――――――――――――――――
   //  SIGNAL         FUNCTION               TYPE     DETAILS
   //  ――――――――――――――――――――――――――――――――――――――――――
   //  Mode_AutMan     Identifies the operating mode of     Bool  1 = automatic mode
   //            the valve.                   0 = manual mode
   //  ――――――――――――――――――――――――――――――――――――――――――
   // 
   // It is possible to configure the module such that manual mode is permanently disabled; this uses 
   // the following STATIC_DATA parameter:
   // 
   //  DATA STRUCTURE    UT11011_St_DevValve3Way
   //  ――――――――――――――――――――――――――――――――――――――――――
   //  SIGNAL         FUNCTION               TYPE     DETAILS
   //  ――――――――――――――――――――――――――――――――――――――――――
   //  CONFIG_MAN_DIS     Prevents manual mode being       Bool  1 = no manual mode
   //            activated under all circumstances            0 = manual permitted
   //            device is in auto, Mode_AutMan is 
   //            set permanently to 1
   //  ――――――――――――――――――――――――――――――――――――――――――
   // 
   // If manual mode is disabled (configuration signal CONFIG_MAN_DIS is set to 1), then manual 
   // mode cannot be turned on under any circumstances, the option will be greyed out on the 
   // supervisory system faceplate and the module will constantly set the mode_AutMan signal to 1.
   // 
   // By default the device will be in automatic mode.
   // 
   // The state of the OPERATE parameter is determined by either the ctrl_Aut_EngDeng or 
   // ctrl_Man_EngDeng, depending on whether automatic mode or manual mode is active. 
   // 
   // The various states of the valve for both automatic and manual operations are given 
   // in the following table:
   // 
   // 
   //  ――――――――――――――――――――――――――――――――――――――――――
   //  MODE:   AUTOMATIC MODE (mode_AutMan = 1)
   //  ctrl_Aut_EngDeng ctrl_Man_EngDeng      OPERATE     VALVE STATE
   //  ――――――――――――――――――――――――――――――――――――――――――
   //      0         N/A          0       Deenergised
   //      1         N/A          1       Energised
   //  ――――――――――――――――――――――――――――――――――――――――――
   //  MODE:   MANUAL MODE (mode_AutMan = 0)
   //  ctrl_Aut_EngDeng ctrl_Man_EngDeng      OPERATE     VALVE STATE
   //  ――――――――――――――――――――――――――――――――――――――――――
   //       N/A          0           0       Deenergised
   //       N/A          1           1       Energised
   //  ――――――――――――――――――――――――――――――――――――――――――
   // 
   // 
   // If the valve is in a fault state (see § 3.4), the OPERATE parameter will be set to 0 (deenergised), 
   // irrespective of any other signals.
   // 
   // 
   // 
   // ▁▁▁▁▁▁▁▁▁▁▁▁▁▁▁▁▁▁▁▁▁▁▁▁▁▁▁▁▁▁▁▁▁▁▁▁▁▁▁▁▁▁▁▁
   // 3.2.2     Operation timers
   // 
   // 
   // The module has an operation timer that is used for both energising and deenergising the valve.
   // 
   // The timer is loaded with either the energising operation time or deenergising operation time 
   // whenever the valve is requested to change state. The timer counts down from the loaded value 
   // to zero (the valve can have different times for energising and deenergising).
   // 
   // The specific operating times are given within the STATIC_DATA parameter 
   // UDT (UT11011_St_DevValve3Way) as follows:
   // 
   // 
   //  DATA STRUCTURE    UT11011_St_DevValve3Way
   //  ――――――――――――――――――――――――――――――――――――――――――
   //  SIGNAL         FUNCTION               TYPE     DETAILS
   //  ――――――――――――――――――――――――――――――――――――――――――
   //  TIME_ENG_MAX    The maximum time required for the     Real     Time in seconds
   //            valve to travel from a deenergised 
   //            state to an energised state
   // 
   //  TIME_DENG_MAX    The maximum time required for the     Real     Time in seconds
   //            valve to travel from an energised 
   //            state to a deenergised state
   //  ――――――――――――――――――――――――――――――――――――――――――
   // 
   // If the timer is running, the elapsed (counting down) time is stored within the DYNAMIC_DATA 
   // parameter UDT (UT31011_Dy_DevValve3Way) as follows:
   // 
   // 
   //  DATA STRUCTURE    UT31011_Dy_DevValve3Way
   //  ――――――――――――――――――――――――――――――――――――――――――
   //  SIGNAL           FUNCTION               TYPE     DETAILS
   //  ――――――――――――――――――――――――――――――――――――――――――
   //  actual_Operating_Timer    The actual elapsed operation time       Real     Time in seconds
   //  ――――――――――――――――――――――――――――――――――――――――――
   // 
   // There is a single operating timer for both energising and deenergising (energising and 
   // deenergising are mutually exclusive operations, hence only one timer is needed. The timer is 
   // preloaded with either the energising time preset or the deenergising time preset prior to the 
   // timer starting).
   // 
   // The preset signals TIME_ENG_MAX and TIME_DENG_MAX are the maximum possible times it can 
   // take for the valve to reach the expected position. This should be set to between 110% and 
   // 120% of the normal energising and deenergising times specified for the valve. For example, if a 
   // valve has a normal energising time of 5 seconds and a normal deenergising time of 3 seconds, 
   // sensible values for TIME_ENG_MAX and TIME_DENG_MAX would be between 5.5-6.0 s and 
   // 3.3-4.0 s respectively.
   // 
   // A valve will enter a fault state (see § 3.4) if the operation timer counts down to a value of zero 
   // without confirmation that the valve has reached the required state. Such confirmation is 
   // provided by positive feedback from the valve limit switches (or other indicating devices) or 
   // by simulated signal within the module itself (see § 3.2.3).
   // 
   // The operation timer always counts down from a preset value to zero, this is in accordance 
   // with the general requirements and practices of the PAL software.
   // 
   // 
   // 
   // ▁▁▁▁▁▁▁▁▁▁▁▁▁▁▁▁▁▁▁▁▁▁▁▁▁▁▁▁▁▁▁▁▁▁▁▁▁▁▁▁▁▁▁▁
   // 3.2.3     Position feedback signals
   // 
   // 
   // The module can accommodate either none, one or two positive position indication signals:
   // 
   //    1.  No limit switches         There is no positive indication of the current state 
   //                      of the valve, it is assumed to be in the expected 
   //                      state.
   // 
   //    2.  Deenergised limit switch only     Positive indication is given for the deenergised 
   //                      state only. The valve is assumed to be in the 
   //                      energised state if the deenergised signal is 
   //                      inactive.
   // 
   //    3.  Energised limit switch only       Positive indication is given for the energised 
   //                      state only. The valve is assumed to be 
   //                      deenergised if the energised signal is inactive.
   // 
   // 
   //    4.  Energised and deenergised        Positive indication is given for both states. 
   //      limit switches            This allows the true state of the valve to be 
   //                      determined under all circumstances.
   // 
   // There are two configuration signals that determine the position feedback arrangements, these 
   // are stored within the STATIC_DATA parameter UDT as follows:
   // 
   // 
   //  DATA STRUCTURE    UT11011_St_DevValve3Way
   //  ――――――――――――――――――――――――――――――――――――――――――
   //  SIGNAL           FUNCTION              TYPE     DETAILS
   //  ――――――――――――――――――――――――――――――――――――――――――
   //  CONFIG_FBK_ENG_EN   Indicates that positive feedback for    Bool  1 = eng feedback
   //              the energised state is present        0 = no feedback
   // 
   //  CONFIG_FBK_DENG_EN   Indicates that positive feedback for    Bool  1 = deng feedback
   //              the deenergised state is present       0 = no feedback
   //  ――――――――――――――――――――――――――――――――――――――――――
   // 
   // If the CONFIG_FBK_ENG_EN signal is activated (set to 1), the module will use the state of the 
   // signal connected to the FBK_ENG parameter to determine the energised position of the valve. 
   // 
   // If the CONFIG_FBK_ENG_EN signal is deactivated (set to 0), the module will derive the 
   // energised position of the valve such that it matches the requested state of the valve.
   // 
   // Similarly, if the CONFIG_FBK_DENG_EN signal is activated (set to 1), the module will use the 
   // state of the signal connected to the FBK_DENG parameter to determine the deenergised 
   // position of the valve. 
   // 
   // If the CONFIG_FBK_DENG_EN signal is deactivated (set to 0), the module will derive the 
   // deenergised position of the valve such that it matches the requested state of the valve.
   // 
   // Where a CONFIG_FBK_ENG/DENG_EN signal is activated (set to 1), a true state on the associated 
   // parameter FBK_ENG/DEENERGISED indicates that the valve is in that position, a false state 
   // indicates that the valve is not in that position as follows:
   // 
   // 
   //  ENERGISED SIGNALS   ――――――――――――――――――――――――――――――――
   //  CONFIG_FBK_ENG_EN       FBK_ENG     MEANING
   //  ――――――――――――――――――――――――――――――――――――――――――
   //       1            0       Not in the energised position
   // 
   //       1            1       Confirmed in the energised position
   // 
   //       0          N/A     Internally derived energised signal matches
   //                        requested valve state, FBK_ENG is ignored
   //  ――――――――――――――――――――――――――――――――――――――――――
   //  DEENERGISED SIGNALS  ―――――――――――――――――――――――――――――――
   //  CONFIG_FBK_DENG_EN       FBK_DENG     MEANING
   //  ――――――――――――――――――――――――――――――――――――――――――
   //       1            0       Not in the deenergised position
   // 
   //       1            1       Confirmed in the deenergised position
   // 
   //       0          N/A     Internally derived deenergised signal matches
   //                        requested valve state, FBK_DENG is ignored
   //  ――――――――――――――――――――――――――――――――――――――――――   
   // 
   // 
   // 
   // 
   // ▁▁▁▁▁▁▁▁▁▁▁▁▁▁▁▁▁▁▁▁▁▁▁▁▁▁▁▁▁▁▁▁▁▁▁▁▁▁▁▁▁▁▁▁
   // Position status signals
   // 
   // 
   // The true position of the valve is given as status signals:
   // 
   //  DATA STRUCTURE    UT31011_Dy_DevValve3Way
   //  ――――――――――――――――――――――――――――――――――――――――――
   //  SIGNAL          FUNCTION               TYPE     DETAILS
   //  ――――――――――――――――――――――――――――――――――――――――――
   //  status_Denergised    Valve is confirmed deenergised      Bool     1 = deenergised
   //                                   0 = not deenergised
   // 
   //  status_Energising     Valve is energising           Bool     1 = energising
   //                                   0 = not energising
   // 
   //  status_Energised      Valve is confirmed energised        Bool     1 = energised
   //                                   0 = not energised
   // 
   //  status_Deenergising   Valve is deenergising         Bool     1 = deenergising
   //                                   0 = not deenergising
   // 
   //  status_Operating      Valve is changing state         Bool     1 = changing state
   //             (either energising                 0 = fixed state
   //              or deenergising)
   // 
   //  status_Fault       Valve is in a fault condition         Bool     1 = fault
   //                                   0 = healthy
   //  ――――――――――――――――――――――――――――――――――――――――――   
   // 
   // 
   // ▁▁▁▁▁▁▁▁▁▁▁▁▁▁▁▁▁▁▁▁▁▁▁▁▁▁▁▁▁▁▁▁▁▁▁▁▁▁▁▁▁▁▁▁
   // Understanding derived position signals
   // 
   // 
   // Where ether the CONFIG_FBK_ENG_EN or CONFIG_FBK_DENG_EN signal is deactivated (set to 0), 
   // the associated position feedback is internally determined by the module according to the actual 
   // state of the valve (determined by the OPERATE parameter)..
   // 
   // These internally derived signals are themselves configurable and can be set such that the 
   // position feedback signal occurs after a particular percentage of the associated operation timer 
   // has expired.
   // 
   // For the derived FBK_ENG signal, the configurable percentage signal is TIME_DER_ENG stored 
   // within the STATIC_DATA parameter. Similarly, for the derived FBK_DENG signal, the configurable 
   // percentage signal is TIME_DER_DENG, again, stored within the STATIC_DATA parameter.
   // 
   // The operation of these parameters can be seen below:
   // 
   //     ①                ③
   // │   ┌────────────────┐
   // │   │                │
   // │   │                │      ctrl_Aut_EngDeng
   // │   │                │
   // ┼───┘┈┈┈┈┈┈┈┈┈┈┈┈┈┈┈┈└───────────────
   // 
   // 
   //                       TIME_ENG_MAX              TIME_DENG_MAX
   //      ←         →       ←                →
   // │   ┌──────┐┄┄┐      ┌───────┐┄┄┐
   // │   │      │  ┆      │       │  ┆
   // │   │←    Ａ  →│  ┆      │←      Ｂ    →│  ┆actual_Operating_Timer
   // │   │      │  ┆      │       │  ┆
   // ┼───┘┈┈┈┈┈┈└──┴──────┘┈┈┈┈┈┈┈└──┴────
   //     ╎      ②         ╎       ④
   //     ╎      ╎         ╎       ╎
   //     ↓      ╎         ╎       ↓
   // │───┐      ╎         ╎       ┌───────
   // │   │      ╎         ╎       │
   // │   │      ╎         ╎       │                FBK_DENG (derived)
   // │   │      ╎         ╎       │
   // ┼┈┈┈└────────────────────────┘┈┈┈┈┈┈┈
   //     Ｃ      ╎         ╎       Ｆ
   //            ╎         ╎
   //            ╎         ╎
   //            ↓         ↓
   // │          ┌─────────┐
   // │          │         │
   // │          │         │               FBK_ENG (derived)
   // │          │         │
   // ┼──────────┘┈┈┈┈┈┈┈┈┈└────────────────
   //            Ｄ         Ｅ
   // 
   //   Ａ TIME_DER_ENG  (90%)
   //   Ｂ TIME_DER_DENG  (80%)
   //   Ｃ Deenergised signal deactivates instantly when the valve is asked to energise
   //   Ｄ Energised signal activates when actual_Operating_Timer reaches TIME_DER_ENG 
   //     as a percentage of TIME_ENG_MAX
   //   Ｅ Energise signal deactivates instantly when the valve is asked to deenergise
   //   Ｆ Deenergised signal activates when actual_Operating_Timer reaches TIME_DER_DENG 
   //     as a percentage of TIME_DENG_MAX
   // 
   // The figure above assumes valve with no position feedback signals (both CONFIG_FBK_ENG_EN 
   // and CONFIG_FBK_DENG_EN are set to 0) operating in automatic mode. It also assumes that the 
   // valve is free to operate without restriction (there are no active interlock or safety signals).
   // 
   // The valve is initially deenergised with the derived FBK_DENG signal active (1) and the derived 
   // FBK_ENG signal deactivated (0). At some point 1, the module receives a request to energised 
   // the valve.
   // 
   // At this point two things happen, firstly the operation timer starts, with a countdown from the value 
   // TIME_ENG_MAX, which in this case is 3 seconds. Secondly, the derived FBK_DENG signal is 
   // deenergised (indicating the valve is no longer deenergised).
   // 
   // The simulated energising time (TIME_DER_ENG) is set to 90%, this means that the derived 
   // FBK_ENG signal will activate when the actual_Operating_Timer value has counted down for 90% 
   // of the TIME_ENG_MAX value (i.e. when the timer has counted down to 0.30s or less). 
   // 
   // The exact formula used is:
   // 
   // 
   // ┌──────────────────────────────────────┐
   // │Derived FBK_ENG = 1 when:                           │
   // │                              TIME_DER_ENG     │
   // │actual_Operating_Timer ≤ TIME_ENG_MAX ─ TIME_ENG_MAX ╳ --------------------------------     │
   // │                                  100      │
   // └──────────────────────────────────────┘
   // 
   // This can be seen at point ②, where the derived FBK_ENG signal activates. The valve now 
   // remains in the energised state (FBK_ENG = 1. FBK_DENG = 0) until there is a request to 
   // deenergise the valve, point ③.
   // 
   // Again, at point ③, the module receives a request to deenergise the valve.
   // 
   // ▁▁▁▁▁▁▁▁▁▁▁▁▁▁▁▁▁▁▁▁▁▁▁▁▁▁▁▁▁▁▁▁▁▁▁▁▁▁▁▁▁▁▁▁
   // At this point two things happen, firstly the operation timer starts, with a countdown from the 
   // value TIME_DENG_MAX, which in this case is 4 seconds. Secondly, the derived FBK_ENG signal is 
   // deenergised (indicating the valve is no longer energised).
   // 
   // The simulated deenergising time (TIME_DER_DENG) is set to 80%, this means that the derived 
   // FBK_DENG signal will activate when the actual_Operating_Timer value has counted down for 
   // 80% of the TIME_DENG_MAX value (i.e. when the timer has counted down to 0.80s or less).  
   // 
   // The exact formula used is:
   // 
   // ┌────────────────────────────────────────┐
   // │Derived FBK_DENG = 1 when:                             │
   // │                               TIME_DER_DENG       │
   // │actual_Operating_Timer ≤ TIME_DENG_MAX ─ TIME_DENG_MAX ╳ ------------------------------------    │
   // │                                  100        │
   // └────────────────────────────────────────┘
   // 
   // This can be seen at point ④, where the derived FBK_DENG signal activates. The valve now 
   // remains in the deenergised state (FBK_ENG = 0. FBK_DENG = 1) until there is a  
   // subsequent request to reenergise the valve.
   // 
   // If only one position feedback is derived (the other being an actual signal), then the derived signal 
   // will be generated in exactly the same way as above, the non-derived signal will simply use the 
   // true status of the signal passed as a parameter to the module.
   // 
   // The simulated time signals are passed to the module within the STATIC_DATA parameter 
   // UDT (UT11011_St_DevValve3Way) as follows:
   // 
   //  DATA STRUCTURE    UT11011_St_DevValve3Way
   //  ――――――――――――――――――――――――――――――――――――――――――
   //  SIGNAL        FUNCTION              TYPE     DETAILS
   //  ――――――――――――――――――――――――――――――――――――――――――
   //  TIME_DER_DENG            Specifies the percentage of the     Real     Percentage
   //              TIME_DENG_MAX value that 
   //              must expire before the derived 
   //              FBK_DENG signal activates.
   // 
   // 
   //  TIME_DER_ENG            Specifies the percentage of the     Real     Percentage
   //              TIME_ENG_MAX value that 
   //              must expire before the derived 
   //              FBK_ENG signal activates.
   //  ――――――――――――――――――――――――――――――――――――――――――
   // 
   // Both configuration signals are restricted to the range 0.00-100.00, the default value is 90% for 
   // both energised and deenergised.
   // 
   // 
   // 
   // ▁▁▁▁▁▁▁▁▁▁▁▁▁▁▁▁▁▁▁▁▁▁▁▁▁▁▁▁▁▁▁▁▁▁▁▁▁▁▁▁▁▁▁▁
   // 3.2.4    Recording the last operation time
   // 
   // 
   // The module records the last complete operation time value, it records the actual time taken for 
   // the valve to reach the correct designated position.
   // 
   // For example if the valve received a request to energise, and it required 4.8 seconds for the 
   // position feedback to report the correct (energised) state, the module would record a value of 
   // 4.8 seconds in the actual_Last_Op_time value (passed as part of the DYNAMIC_DATA parameter).
   // 
   // Similarly, if the valve were requested to deenergise, and required 6.2 seconds for the position 
   // feedback to report the correct (deenergised) state, the module would record a value of 
   // 6.2 seconds in the actual_Last_Op_time value..
   // 
   // The actual_Last_Op_time value forms part of the DYNAMIC_DATA parameter UDT as follows:
   // 
   // 
   //  DATA STRUCTURE    UT31011_Dy_DevValve3Way
   //  ――――――――――――――――――――――――――――――――――――――――――
   //  SIGNAL        FUNCTION              TYPE     DETAILS
   //  ――――――――――――――――――――――――――――――――――――――――――
   //  actual_Last_Op_Time     Stores the actual time taken for     Real     Time in seconds
   //             the valve to achieve the correct 
   //             energised or deenergised state.
   // 
   //             Receives a value of -1.0 if the 
   //             valve did not achieve the correct 
   //             position in the specified 
   //             operation time
   //  ――――――――――――――――――――――――――――――――――――――――――
   // 
   // If the valve does not achieve the requested position (within either the TIME_ENG_MAX or 
   // TIME_DENG_MAX limits), a value of -1.0 is returned as the actual_Last_Op_time value, indicating 
   // a fault occurred.
   // 
   // 
   // 
   // ▁▁▁▁▁▁▁▁▁▁▁▁▁▁▁▁▁▁▁▁▁▁▁▁▁▁▁▁▁▁▁▁▁▁▁▁▁▁▁▁▁▁▁▁
   // 3.2.5    Detecting position faults
   // 
   // 
   // There are two types of position faults: dynamic and static. 
   // 
   // Dynamic faults occur when the valve is changing state (from energised to deenergised or 
   // deenergised to energised) and fails to achieve the requested position within the relevant 
   // operation time.
   // 
   // The dynamic faults are:
   // 
   //    •   Failed to energise
   // 
   //    •   Failed to deenergise
   // 
   // Static faults occur when a valve is stable in the requested state (either energised or 
   // deenergised) and is not in the process of moving between states, and some fault occurs such 
   // that the position feedback no longer matches the requested state (e.g. the valve was correctly 
   // in the energised state, and then at some point, the energised feedback signal was lost without 
   // any change being made to the state of the valve by the module. Such a fault could be a power 
   // failure at the valve).
   // 
   // The static faults are:
   // 
   //    •   Failed while energised
   // 
   //    •   Failed while deenergised
   // 
   // If the valve is not equipped with any limit switches (both CONFIG_FBK_ENG_EN and 
   // CONFIG_FBK_DENG_EN are set to 0), then there are no circumstances under which any position 
   // fault can be generated (the valve is always assumed to operate correctly and be in the 
   // required position). 
   // 
   // The following table indicates the conditions under which the various alarms can be generated 
   // for the various position feedback combinations:
   // 
   //  ――――――――――――――――――――――――――――――――――――――――――
   //                   FAILED TO ENERGISE         FAILED TO DEENERGISE
   //        LIMIT SWITCH      Energising operation timer     Deenergising operation timer 
   //      ARRANGEMENT        expired and:                 expired and:
   //  ――――――――――――――――――――――――――――――――――――――――――
   //        No feedback
   //      CONFIG_FBK_ENG_EN = 0     Not applicable         Not applicable
   //    CONFIG_FBK_DENG_EN = 0
   // 
   //      Energised feedback only
   //      CONFIG_FBK_ENG_EN = 1   Energised feedback      Energised feedback
   //    CONFIG_FBK_DENG_EN = 0       is INACTIVE            is ACTIVE
   // 
   //   Deenergised feedback only
   //      CONFIG_FBK_ENG_EN = 0    Deenergised feedback       Deenergised feedback
   //    CONFIG_FBK_DENG_EN = 1         is ACTIVE             is INACTIVE
   // 
   //      Both feedback     Deenergised feedback ACTIVE  Deenergised feedback INACTIVE
   //      CONFIG_FBK_ENG_EN = 1         OR                   OR
   //    CONFIG_FBK_DENG_EN = 1   Energised feedback INACTIVE  Energised feedback is ACTIVE
   //  ――――――――――――――――――――――――――――――――――――――――――
   // 
   //  ――――――――――――――――――――――――――――――――――――――――――
   //                 FAILED WHILE ENERGISED     FAILED WHILE ENERGISED
   //        LIMIT SWITCH      Energising operation timer     Deenergising operation timer 
   //      ARRANGEMENT        not running and:        not running and:
   //  ――――――――――――――――――――――――――――――――――――――――――
   //        No feedback
   //      CONFIG_FBK_ENG_EN = 0     Not applicable         Not applicable
   //    CONFIG_FBK_DENG_EN = 0
   // 
   //      Energised feedback only
   //      CONFIG_FBK_ENG_EN = 1   Energised feedback      Energised feedback
   //    CONFIG_FBK_DENG_EN = 0       is INACTIVE            is ACTIVE
   // 
   //   Deenergised feedback only
   //      CONFIG_FBK_ENG_EN = 0    Deenergised feedback       Deenergised feedback
   //    CONFIG_FBK_DENG_EN = 1         is ACTIVE             is INACTIVE
   // 
   //      Both feedback     Deenergised feedback ACTIVE  Deenergised feedback INACTIVE
   //      CONFIG_FBK_ENG_EN = 1         OR                   OR
   //    CONFIG_FBK_DENG_EN = 1   Energised feedback INACTIVE  Energised feedback is ACTIVE
   //  ――――――――――――――――――――――――――――――――――――――――――
   // 
   // The OR in the alarm conditions is a logical or, it covers the conditions in which both or neither 
   // limit switches are active; consider the failed to energised alarm, if both limits were active, the 
   // alarm would be generated because the deenergised limit switch is active (irrespective of the 
   // state of the energised limit). Similarly, if neither switch were active, the alarm would be 
   // generated because the energised limit is inactive (irrespective of the state of the deenergised 
   // limit).
   // 
   // All alarms are reported as message signals, these form part of the DYNAMIC_DATA parameter 
   // UDT as follows:
   // 
   //  DATA STRUCTURE    UT31011_Dy_DevValve3Way
   //  ――――――――――――――――――――――――――――――――――――――――――
   //  SIGNAL          FUNCTION                TYPE     DETAILS
   //  ――――――――――――――――――――――――――――――――――――――――――
   //  msg_FailToEnergise       Valve failed to energise in the     Bool     1 = alarm active
   //               specified energising time             0 = no alarm
   // 
   //  msg_FailToDeenergise     Valve failed to deenergise in the   Bool     1 = alarm active
   //               specified deenergising time            0 = no alarm
   // 
   //  msg_FailWhileEnergised     Valve suffered position failure     Bool     1 = alarm active
   //               while in a static ENERGISED state         0 = no alarm
   // 
   //  msg_FailWhileDeenergised   Valve suffered position failure     Bool     1 = alarm active
   //               while in a static DEENERGISED state       0 = no alarm
   //  ――――――――――――――――――――――――――――――――――――――――――
END_REGION

REGION Network 3: Block description — Section 3.3 to 3.5
   // ▂▂▂▂▂▂▂▂▂▂▂▂▂▂▂▂▂▂▂▂▂▂▂▂▂▂▂▂▂▂▂▂▂▂▂▂▂▂▂▂▂▂▂▂
   // 3.3     Fault handling
   // 
   // 
   // There are five fault conditions, four are derived from position faults and one from an external 
   // fault signal:
   // 
   //  ――――――――――――――――――――――――――――――――――――――――――
   //  FAULT           DESCRIPTION                  LATCHING
   //  ―――――――――――――――――――――――――――――――――――――――――― 
   //  Failed to energise       Valve failed to reach the energise state in       YES
   //               the specified energising operation time
   // 
   //  Failed to deenergise      Valve failed to deenergise state in            YES
   //               the specified deenergising operation time
   // 
   //  Failed while energised     Valve suffered position failure while          YES
   //               in a static ENERGISED state
   // 
   //  Failed while deenergised   Valve suffered positions failure while        YES
   //               in a static DEENERGISED state
   // 
   //  External fault          The EXT_FAULT signal is active           NO
   //   ――――――――――――――――――――――――――――――――――――――――――
   // 
   // If any of the above faults are active, the valve will be deenergised (the OPERATE parameter will be 
   // set to 0) and the module will ignore all commands either automatic or manual and will ignore all 
   // interlock conditions.
   // 
   // 
   // ▁▁▁▁▁▁▁▁▁▁▁▁▁▁▁▁▁▁▁▁▁▁▁▁▁▁▁▁▁▁▁▁▁▁▁▁▁▁▁▁▁▁▁▁
   // 3.3.1    Position faults
   // 
   // 
   // All position faults (derived from position feedback signals) are latching fault conditions that  
   // require the operator to issue a reset command, this is usually via a faceplate available at the 
   // supervisory system (SCADA/HMI), but could also be via a hardwired 
   // (pushbutton) signal. 
   // 
   // The reset signal is specified within the DYNAMIC_DATA parameter UDT as follows:        
   // 
   //  DATA STRUCTURE    UT31011_Dy_DevValve3Way
   //  ――――――――――――――――――――――――――――――――――――――――――
   //  SIGNAL         FUNCTION                TYPE     DETAILS
   //  ――――――――――――――――――――――――――――――――――――――――――
   //  mode_Reset        A reset pulse                Bool     1 = reset latched faults
   //            (active for one Controller cycle)            0 = no action
   //  ――――――――――――――――――――――――――――――――――――――――――
   // 
   // 
   // 
   // ▁▁▁▁▁▁▁▁▁▁▁▁▁▁▁▁▁▁▁▁▁▁▁▁▁▁▁▁▁▁▁▁▁▁▁▁▁▁▁▁▁▁▁▁
   // 3.3.2    Resetting position faults
   // 
   // 
   // If a position fault has occurred, and the fault is then reset, the appropriate energising or 
   // deenergising operation timer will be retriggered, allowing the valve time to achieve the required 
   // position.
   // 
   // 
   // 
   // ▁▁▁▁▁▁▁▁▁▁▁▁▁▁▁▁▁▁▁▁▁▁▁▁▁▁▁▁▁▁▁▁▁▁▁▁▁▁▁▁▁▁▁▁
   // 3.3.3    External fault
   // 
   // 
   // The external fault is an optional hardwired signal from the valve, it indicates that the device 
   // itself is registering that there is some problem. Such external fault signals are more commonly 
   // associated with motorised valves (equipped with thermal overload detectors), but may also be 
   // associated with pneumatic or hydraulic operated valves to indicate that the is a 
   // pneumatic/hydraulic system failure.
   // 
   // Such fault signals are generally indicated via a hardwired digital input to the Controller.
   // 
   // The external fault signal (if used) is passed to the module as the parameter: EXT_FAULT .
   // 
   // Any signal connected to the EXT_FAULT parameter must be active high (i.e. the signal must be 
   // set to 1 to indicate the fault condition is present). 
   // 
   // Where a failsafe response signal is used (active when set to 0) is used, it must be inverted at the 
   // EXT_FAULT parameter:
   // 
   //                         ┌─────────────
   //      ───────────────────┤ FC11011 
   //                         ├───────────────┤
   //           "V001_FAULT"                  │               │
   //        ────┤╱├──────────┤ EXT_FAULT             │
   //                         │               
   //                         │               
   // 
   // If the EXT_FAULT signal is not required, the input should be set to _False  (again, similar to the
   // E_STOP signal).
   // 
   // The EXT_FAULT signal is non-latching; it does not require a mode_Reset signal to clear the fault. 
   // The external fault will automatically reset whenever the EXT_FAULT signal is set to 0.
   // 
   // 
   // 
   // ▂▂▂▂▂▂▂▂▂▂▂▂▂▂▂▂▂▂▂▂▂▂▂▂▂▂▂▂▂▂▂▂▂▂▂▂▂▂▂▂▂▂▂▂
   // 3.4     Safety and interlocks
   // 
   // 
   // Safety and interlock signals are optional signals, passed as individual parameters to the module 
   // (in the same a manner as IO signals), all such signals are optional, a valve can have all, none or 
   // any combination of the signals.
   // 
   // Safety and interlock signals all act to override the normal operation of the valve (whether in 
   // automatic or manual mode) and force the valve to a particular state.
   // 
   // There is one safety signal and three interlock signals, each having its own formal module 
   // parameter:
   // 
   // 
   //  SAFETY SIGNAL
   //  ――――――――――――――――――――――――――――――――――――――――――
   //  PARAM        FUNCTION                   TYPE     DETAILS 
   //  ――――――――――――――――――――――――――――――――――――――――――
   //  E_STOP       Optional emergency stop (safety) signal       Bool     1 = E-stop active
   //          (1 = emergency stop active, 0 = healthy) If not         0 = healthy
   //          required, set permanently to _False
   //  ――――――――――――――――――――――――――――――――――――――――――
   // 
   // 
   //  INTERLOCK SIGNALS
   //  ――――――――――――――――――――――――――――――――――――――――――
   //  PARAM        FUNCTION                   TYPE     DETAILS  
   //  ――――――――――――――――――――――――――――――――――――――――――
   //  TRIP       Optional trip signal                 Bool     1 = Trip active
   //          (1 = trip condition active, 0 = healthy) If not            0 = healthy
   //          required, set permanently to _False
   // 
   //  INTERLOCK    Optional interlock signal              Bool     1 = Interlock active
   //          (1 = interlock condition active, 0 = healthy) If         0 = healthy
   //          not required, set permanently to _False
   // 
   //  PERMISSIVE     Optional permissive signal            Bool     1 = Permissive active
   //          (1 = permissive condition active, 0 = healthy)           0 = healthy
   //          If not required, set permanently to _False
   //  ――――――――――――――――――――――――――――――――――――――――――
   // 
   // 
   // Each safety and interlock signal has its own configuration signal that must be used to formally 
   // disable the parameter if the signal is not required, these are all within the STATIC_DATA parameter 
   // UDT (UT11011_St_DevValve3Way) as follows:
   // 
   // 
   //  DATA STRUCTURE    UT11011_St_DevValve3Way
   //  ――――――――――――――――――――――――――――――――――――――――――
   //  SIGNAL        FUNCTION              TYPE     DETAILS
   //  ――――――――――――――――――――――――――――――――――――――――――
   //  CONFIG_ESTOP_DIS    Disables the safety signal.        Bool     1 = E_STOP disabled
   //              If set to 1, any signal on the          0 = E_STOP enabled
   //              E_STOP parameter will be 
   //              ignored.
   // 
   //  CONFIG_TRIP_DIS      Disables the trip interlock signal.   Bool     1 = TRIP disabled
   //              If set to 1, any signal on the          0 = TRIP enabled
   //              TRIP parameter will be 
   //              ignored.
   // 
   //  CONFIG_ILOCK_DIS     Disables the interlock signal.    Bool     1 = INTERLOCK disabled
   //              If set to 1, any signal on the          0 = INTERLOCK enabled
   //              INTERLOCK parameter will be 
   //              ignored.
   // 
   //  CONFIG_PERM_DIS   Disables the permissive interlock  Bool     1 = PERMISSIVE disabled
   //              signal. If set to 1, any signal on the       0 = PERMISSIVE enabled
   //              TRIP parameter will be 
   //              ignored.
   //  ――――――――――――――――――――――――――――――――――――――――――
   // 
   // The disable signals are used to formally configure the valve, they allow any supervisory system to 
   // know the correct configuration of the valve and display information accordingly.
   // 
   // 
   // 
   // ▁▁▁▁▁▁▁▁▁▁▁▁▁▁▁▁▁▁▁▁▁▁▁▁▁▁▁▁▁▁▁▁▁▁▁▁▁▁▁▁▁▁▁▁
   // 3.4.1    Safety signal operation
   // 
   // 
   // Safety or emergency stop signals are hardwired signals that remove power from a device forcing 
   // it to a safe state. Such signals act independently of the software (the pressing of an emergency 
   // stop button will physically remove power from the affected devices).
   // 
   // The emergency stop signal is passed to the module as the parameter E_STOP; it informs the 
   // module that the safety signal has been activated and allows the module to adjust the state of 
   // the valve to follow the emergency stop conditions.
   // 
   // When the emergency stop signal is removed, the valve will resume the requested state (with the 
   // appropriate operation timer).
   // 
   // Under emergency stop conditions the valve is always deenergised (both physically by the 
   // hardware and within the software via the actions of this module), the OPERATE output is set to 
   // zero (OPERATE = 0).
   // 
   // The emergency stop signal is absolute and will override any other demand made of the valve. 
   // There is no mechanism for bypassing this form of safety signal.
   // 
   // 
   // 
   // ▁▁▁▁▁▁▁▁▁▁▁▁▁▁▁▁▁▁▁▁▁▁▁▁▁▁▁▁▁▁▁▁▁▁▁▁▁▁▁▁▁▁▁▁
   // Typical usage of the E_STOP parameter
   // 
   // 
   // Any safety signal connected to the E_STOP parameter must be active high (i.e. the signal must be 
   // set to 1 to activate the safety signal response). It is often the case, where hardwired emergency 
   // stop signals are used, that the emergency stop condition is activated by the absence of a signal 
   // (a failsafe response) rather than the application of a signal. The module can accommodate this 
   // sense of signal by inverting the E_STOP input:
   // 
   // 
   //                         ┌─────────────
   //      ───────────────────┤ FC11011 
   //                         ├───────────────┤
   //           "ZONEA_ESTOP"              │               │
   //        ────┤╱├──────────┤ E_STOP             │
   //                         │               
   //                         │               
   // 
   // 
   // If no safety signal is used, the parameter is set to the _False tag (note, also that the configuration 
   // signal CONFIG_ESTOP_DIS should also be set to 1):
   // 
   // 
   //                         ┌─────────────
   //      ───────────────────┤ FC11011 
   //                         ├───────────────┤
   //                         │               │
   //                      _False ──┤ E_STOP             │
   //                         │               
   //                         │    
   // 
   // 
   // 
   // ▁▁▁▁▁▁▁▁▁▁▁▁▁▁▁▁▁▁▁▁▁▁▁▁▁▁▁▁▁▁▁▁▁▁▁▁▁▁▁▁▁▁▁▁
   // 3.4.2    Interlock signals
   // 
   // 
   // Interlock signals are a more flexible mechanism for overriding the requested position of the valve. 
   // Interlock signals can be both hardware driven (similar to a safety signal) or can be purely software 
   // derived (unlike a safety signal).
   // 
   // Software derived interlock signals can accommodate more complex and more flexible 
   // arrangements, it would for example, be possible to disable a software derived interlock if the 
   // process were undergoing some particular function, such as cleaning &c.
   // 
   // There are three different types of interlock arrangements:
   // 
   // There are three types of interlock signal:
   // 
   //    1.  INTERLOCK
   //      A simple interlock that is active whenever a set of conditions is true, it will force any 
   //      associated devices to a given safe state.
   // 
   //    2.  PERMISSIVE
   //      Takes no action if a device is in a non-safe state, but once the device is in a safe 
   //      state will prevent a transition to a non-safe state (i.e. will not force a valve to 
   //      deenergise, but once it is deenergised will prevent it from re-energising).
   // 
   //    3.  TRIP
   //      A latching interlock, it activates whenever a set of events are true (like an interlock), 
   //      but will not deactivate until the triggering conditions are removed and a reset signal 
   //      has been given (effectively a latching interlock), it will force any associated devices 
   //      to a given safe state.
   // 
   // For any type of interlock, the specified interlock state (or permitted state) can be either 
   // energised or deenergised; unlike the safety signal, it does not have to be the deenergised state 
   // of the valve.
   // 
   // That said, the most common interlock state is the deenergised state of the valve; i.e. the failsafe 
   // position of the valve.
   // 
   // 
   // 
   // ▁▁▁▁▁▁▁▁▁▁▁▁▁▁▁▁▁▁▁▁▁▁▁▁▁▁▁▁▁▁▁▁▁▁▁▁▁▁▁▁▁▁▁▁
   // Typical usage of interlock signals
   // 
   // 
   // Each type of interlock is passed as its own parameter: TRIP, INTERLOCK or PERMISSIVE. Like the 
   // safety signal (E_STOP), each parameter is active high (i.e. the signal must be set to 1 to activate 
   // the associated interlock signal response). 
   // 
   // Again, it is often the case, where hardwired interlock signals are used, that the condition is 
   // activated by the absence of a signal (i.e. a failsafe response) rather than the application of a 
   // signal. The module can accommodate this sense of signal by inverting the relevant input:
   // 
   // 
   //                         ┌─────────────
   //      ───────────────────┤ FC11011 
   //                         ├───────────────┤
   //        "DB23102_Dy_Perm.V001"     │               │
   //        ────┤╱├──────────┤ PERMISSIVE           │
   //                         │               
   // 
   // If a particular interlock signal is not used, the parameter is set to the _False tag (note also: that 
   // the appropriate configuration signal should also be set to 1: CONFIG_TRIP_DIS, CONFIG_ILOCK_DIS 
   // or CONFIG_PERM_DIS).
   // 
   //                         ┌─────────────
   //      ───────────────────┤ FC11011 
   //                         ├───────────────┤
   //                         │               │
   //                      _False ──┤ TRIP                    │
   //                         │               
   //                         │  
   // 
   // 
   // 
   // ▁▁▁▁▁▁▁▁▁▁▁▁▁▁▁▁▁▁▁▁▁▁▁▁▁▁▁▁▁▁▁▁▁▁▁▁▁▁▁▁▁▁▁▁
   // Configuring the interlock signals
   // 
   // 
   // The state adopted by the valve when a particular interlock is active (TRIP or INTERLOCK) or the 
   // permitted state of the valve (PERMISSIVE) are set individually for each type of interlock signal. 
   // These configuration signals are stored within the STATIC_DATA parameter UDT as follows:
   // 
   // 
   //  DATA STRUCTURE    UT11011_St_DevValve3Way
   // 
   //  ――――――――――――――――――――――――――――――――――――――――――
   //  SIGNAL         FUNCTION              TYPE    DETAILS
   //  ――――――――――――――――――――――――――――――――――――――――――
   //  CONFIG_TRIP_ENG_DENG  The required state of a valve if     Bool     1 = will energise
   //               the TRIP signal is active            0 = will deenergise
   // 
   //  CONFIG_ILOCK_ENG_DENG The required state of a valve if     Bool     1 = will energise
   //               the INTERLOCK signal is active         0 = will deenergise
   // 
   //  CONFIG_PERM_ENG_DENG  The permitted state of a valve if     Bool     1 = may energise
   //               the PERMISSIVE signal is active           0 = may deenergise
   //  ――――――――――――――――――――――――――――――――――――――――――
   // 
   // For example, if CONFIG_ILOCK_ENG_DENG is set to 1, the valve will energise whenever the 
   // INTERLOCK signal is active (set to 1), this will override any automatic or manual requirement for 
   // the valve (but will not override a safety signal, see below). If CONFIG_ILOCK_ENG_DENG were set 
   // to 0, the valve would deenergise whenever the INTERLOCK signal was active.
   // 
   // The TRIP signal behaves in exactly the same way as the INTERLOCK signal, but uses 
   // CONFIG_TRIP_ENG_DENG to set the tripped state of the valve.
   // 
   // Although the TRIP signal requires a reset signal to disengage the interlock conditions, this is 
   // handled by the trip logic itself (usually handled by the trip application modules: FC23200) and 
   // not via this module; simply deactivating the TRIP signal removes the trip state from the valve 
   // and allows it to operate normally.
   // 
   // The PERMISSIVE signal operates in a different way, if CONFIG_PERM_ENG_DENG were set to 1 
   // (valve is permitted to be energised), and the valve was currently deenergised under automatic 
   // control when the PERMISSIVE signal became active, nothing would happen to the valve (it would 
   // remain deenergised), if the valve was then subsequently energised under automatic control, 
   // the PERMISSIVE signal would allow the valve to do so (the valve permitted state is energised). 
   // However, any attempt by the automatic system to then deenergised the valve would not be 
   // allowed by the PERMISSIVE signal.
   // 
   // Conversely, if CONFIG_PERM_ENG_DENG were set to 0 (valve is permitted to be deenergised), and 
   // the valve was currently energised under automatic control when the PERMISSIVE signal became 
   // active, nothing would happen to the valve (it would remain energised), if the valve was then 
   // subsequently deenergised under automatic control, the PERMISSIVE signal would allow the 
   // valve to do so (the valve permitted state is deenergised). However, any attempt by the 
   // automatic system to re-energised the valve would not be allowed by the PERMISSIVE signal.
   // 
   // Note:    Where multiple interlock signals are used, it is possible for the different interlocks 
   //      to apply different states to the valve, for example an active TRIP could deenergised 
   //      the valve and an active INTERLOCK energised it. Such conflicts are managed by the 
   //      different priorities applied to the interlock signals (see § 3.5). 
   // 
   // 
   // 
   // ▁▁▁▁▁▁▁▁▁▁▁▁▁▁▁▁▁▁▁▁▁▁▁▁▁▁▁▁▁▁▁▁▁▁▁▁▁▁▁▁▁▁▁▁
   // Bypassing interlocks
   // 
   // 
   // Unlike safety signals, all interlock signals can be overridden (or bypassed). The bypass signal is a 
   // single signal that, if active, overrides and deactivates any TRIP, INTERLOCK or PERMISSIVE signal 
   // that may have been activated.
   // 
   // The bypass signal is specified within the DYNAMIC_DATA parameter UDT as follows:
   // 
   // 
   //  DATA STRUCTURE    UT31011_Dy_DevValve3Way
   //  ――――――――――――――――――――――――――――――――――――――――――
   //  SIGNAL         FUNCTION                TYPE     DETAILS
   //  ――――――――――――――――――――――――――――――――――――――――――
   //  mode_BypassOn   Activates bypass mode, if active, any    Bool     1 = bypass mode on
   //            TRIP, INTERLOCK or PERMISSIVE signal          0 = bypass mode off
   //            will be ignored
   //  ――――――――――――――――――――――――――――――――――――――――――
   // 
   // 
   // Bypass mode is a manual operation, generally activated by the operator via a faceplate 
   // available at the supervisory system (SCADA/HMI), or via some hardwired signal, such as 
   // a key-switch.
   // 
   // It is possible to configure the module such that bypass mode is permanently disabled, this uses 
   // the following STATIC_DATA parameter:
   // 
   // 
   //  DATA STRUCTURE    UT11011_St_DevValve3Way
   //  ――――――――――――――――――――――――――――――――――――――――――
   //  SIGNAL       FUNCTION                TYPE     DETAILS
   //  ――――――――――――――――――――――――――――――――――――――――――
   //  CONFIG_BYPASS_DIS    Prevents bypass mode being      Bool     1 = no bypass mode
   //             activated under all circumstances         0 = bypass permitted
   //  ――――――――――――――――――――――――――――――――――――――――――
   //   
   // If bypass mode is disabled (configuration signal CONFIG_BYPASS_DIS is set to 1), then the bypass 
   // mode cannot be turned on under any circumstances, the option will be greyed out on the 
   // supervisory system faceplate and the module will constantly reset the mode_BypassOn signal.
   // 
   // Note:    Safety (E_STOP) signals cannot be bypassed.  
   // 
   //      Similarly, if an interlock signal has a hardwired component (that will override any 
   //      software actions), it also must not be bypassed.
   // 
   // 
   // 
   // ▂▂▂▂▂▂▂▂▂▂▂▂▂▂▂▂▂▂▂▂▂▂▂▂▂▂▂▂▂▂▂▂▂▂▂▂▂▂▂▂▂▂▂▂
   // 3.5     Priority of operation
   // 
   // 
   // The valve is normally controlled by either the automatic system or by manual (operator) control; 
   // however, this operation can be overridden by the various safety and interlock conditions 
   // that can apply to the valve. Each of these operations is assigned a priority and if more than one 
   // is active at the same time, the one with the highest priority will take precedence.
   // 
   // The priorities for the various operations is as follows:
   // 
   // 
   //  ――――――――――――――――――――――――――――――――――――――――――
   //  SIGNAL TYPE       PRIORITY   ASSIGNED VALUE       CAN BE BYPASSED
   //  ――――――――――――――――――――――――――――――――――――――――――
   //  Emergency Stop        High        40                NO
   //  Trip            ↑           30             YES
   //  Interlock            ↑           20             YES
   //  Permissive          ↑           10             YES
   //  Auto/manual control    Low         00                NO
   //  ――――――――――――――――――――――――――――――――――――――――――
   //  High priority signal take precedence over lower priority signals.
   // 
   // Thus, if both the TRIP signal, the INTERLOCK signal and automatic control signal were all active at 
   // the same time, the module will respond only to the TRIP signal (with the higher priority) and will 
   // react accordingly.
END_REGION

